(*
--报错编号0: 无报错
--报错编号1: openend Error
--报错编号2: closeract Error
*)
FUNCTION_BLOCK MFCModule
VAR_IN_OUT
	WarmHMI					:WARMStruct;
	operatorLog				:printLogModule_EX;
END_VAR
VAR_INPUT
	MFCType						:MFCType:=MFCType_Default;// 设置MFC的类型
	MFCHMItif					:MFCStruct;
	set							:BOOL:=FALSE;// 设置触发信号
	setCondition				:BOOL:=TRUE;// 设置触发条件
	clear						:BOOL:=FALSE;// 清零触发信号
	clearCondition				:BOOL:=TRUE;// 清零条件
	reset						:BOOL:=FALSE;// 复位信号
	stop						:BOOL:=FALSE;// 停止信号
	power						:BOOL:=TRUE;// TRUE--保持得电,FALSE--断开得电
	enable						:BOOL:=TRUE;// MFC禁用条件
	//ctrlMode					:ControlMode:=ControlMode.eManualCtrMode;//eManualCtrMode or eAutoCtrMode
	hmiEN						:BOOL:=TRUE;//HMI 启用条件
	
	errorDelayTime				:TIME:=T#2S;// MFC设置参数超时
	
	ACCMaxtime					:TIME:=T#2S;// MFC加速最大时间
	DCCMaxtime					:TIME:=T#2S;// MFC减速最大时间
	
	doneDelayTimeShortset		:TIME:=T#10MS;// MFC设置值到达延时_设置
	doneDelayTimeShortclear		:TIME:=T#10MS;// MFC设置值到达延时_清零
	errorID						:UDINT:=0;// MFC错误报警分配的起始ID
	nameTXT						:STRING(255):='';// MFC名字
	
	AlmAprSw					:BOOL:=FALSE;// 分子泵报警感应器信号,需要链接到实际的IO点
	
	temperatureMax				:REAL;// MFC温度报警设置值
	setFlow						:UDINT;// MFC流量设定
	maxSetValue					:REAL;// MFC流量设定上限
	minSetValue					:REAL;// MFC流量设定下限
	serialSlaveID				:UINT;// MFC ID
	serialError					:BOOL;// MFC通讯错误
	noteWTXT_set				:WSTRING(255):="";// MFC设置动作NoteTXT 中文
	noteWTXT_clear				:WSTRING(255):="";// MFC清零动作NoteTXT 中文
	
	serialExcute				:BOOL;// 通讯数据发送
	connected					:BOOL;
	connectedCount				:UDINT;
	flow					:UDINT;// 设定反馈流量值
	
	actflow					:UDINT;// 实际反馈流量值
	actflowFloat			:REAL;// 实际反馈流量值
END_VAR
VAR_OUTPUT
	note_set				:BOOL;// 设置条件不满足提示
	note_clear				:BOOL;// 清零条件不满足提示
	
	sendBusy				:BOOL;// 串口发送数据繁忙
	
	busy					:BOOL;// MFC动作Busy状态
	setbusy					:BOOL;// MFC设置动作Busy状态
	clearbusy				:BOOL;// MFC清零动作Busy状态
	done					:BOOL;// MFCdone状态
	setdone					:BOOL;// MFC设置完成
	cleardone				:BOOL;// MFC清零完成
	error					:BOOL;//  MFC error状态
	errID					:UDINT;// MFC errID
	errTXT					:STRING(255):='';//  MFC errTXT
	errWTXT					:WSTRING(255):="";//  MFC errTXT 中文
END_VAR
	
VAR	
	setErrorDelayTon		:Ton;
	setDoneDelayTon			:Ton;
	clearErrorDelayTon		:Ton;
	clearDoneDelayTon		:Ton;
	
	setTrigRAlc			    :R_Trig;//上升沿触发
	
	clearTrigRAlc			:R_Trig;//上升沿触发
	
	setTrigR1			:R_Trig;//上升沿触发
	setTrigR1_Aiko		:R_Trig;//上升沿触发
	clearRactTrigR1			:R_Trig;//上升沿触发
	resetTrigR1				:R_Trig;//上升沿触发
	stopTrigR1				:R_Trig;//上升沿触发
	powerTrigR1				:R_Trig;//上升沿触发
	
	setStep					:UINT:=0;
	clearStep				:UINT:=0;
	errorStep				:UINT:=0;
	
	resetRelayTON			:TON;
	resetRelayTONTime		:TIME:=T#2S;
	
	AccFTrig:F_TRIG;//检测加速信号下降延
	DccFTrig:F_TRIG;// 检测减速信号下降延
	noteTON_P:tON;            // 操作提示标志位延时继电器
	noteTON_N:tON;            // 操作提示标志位延时继电器
	noteRTrig_P:R_TRIG;          // 操作提示
	noteRTrig_N:R_TRIG;          // 操作提示
END_VAR

Init_ACT();
Error_ACT();
Set_ACT();
Clear_ACT();
Reset_ACT();
Error_ACT();

(*
触发缩回动作，成功触发返回TRUE，触发失败返回FALSE
*)
METHOD Act_Clear : BOOL
VAR_INPUT
END_VAR
IF enable AND clearCondition THEN// AND NOT busy
	Act_Clear:=clear:=TRUE;
ELSE
	Act_Clear:=FALSE;
END_IF
END_METHOD

(*
触发复位报警动作，成功触发返回TRUE，触发失败返回FALSE
*)
METHOD Act_Reset : BOOL
VAR_INPUT
END_VAR
Act_Reset:=reset:=TRUE;
END_METHOD

(*
触发发送动作，成功触发返回TRUE，触发失败返回FALSE
*)
METHOD Act_SerialSend : BOOL
VAR_INPUT
END_VAR
IF TRUE THEN
	Act_SerialSend:=serialExcute:=TRUE;
ELSE
	Act_SerialSend:=FALSE;
END_IF
END_METHOD

(*
触发伸出动作，成功触发返回TRUE，触发失败返回FALSE
*)
METHOD Act_Set : BOOL
VAR_INPUT
	_setpoint:UDINT;
END_VAR
IF enable AND setCondition THEN// AND NOT busy
	setFlow:=_setpoint;
	Act_Set:=set:=TRUE;
ELSE
	Act_Set:=FALSE;
END_IF
END_METHOD

(*
触发停止输出动作，成功触发返回TRUE，触发失败返回FALSE
*)
METHOD Act_Stop : BOOL
VAR_INPUT
END_VAR
Act_Stop:=stop:=TRUE;
END_METHOD

ACTION Clear_ACT:
//MFC--clear 触发
IF clear AND NOT clearCondition THEN
	note_set:=FALSE;
	note_clear:=TRUE;
END_IF
IF clear AND enable AND NOT error AND clearCondition AND NOT clearbusy AND NOT gMFCStopLoopRead THEN// AND NOT busy
	note_set:=FALSE;
	note_clear:=FALSE;
	busy:=TRUE;
	clearbusy:=TRUE;
	setbusy:=FALSE;
	set:=FALSE;
	setdone:=FALSE;
	cleardone:=FALSE;
	setStep:=0;
	clearStep:=10;
	gMFCStopLoopRead:=TRUE;
	operatorLog.append(CONCAT(nameTXT,' Clear'));
	//errorStep:=0;
END_IF
clear:=FALSE;

CASE clearStep OF
0:
	//ready
	
10:
	IF FuncModule_RS485_MFC.loopReadStep<10 OR FuncModule_RS485_MFC.loopReadStep>270 THEN
		clearErrorDelayTon(IN:=FALSE);
		clearDoneDelayTon(IN:=FALSE);
		clearStep:=20;
		setFlow:=0;
		FuncModule_RS485_MFC.Interface_Set(serialSlaveID,setFlow);
	END_IF
	
20:
	clearErrorDelayTon(IN:=(NOT FuncModule_RS485_MFC.setDone ),PT:=errorDelayTime);
	IF clearErrorDelayTon.Q THEN
		//done:=FALSE;
		setdone:=FALSE;
		cleardone:=FALSE;
		errorStep:=2;
		clearStep:=60;
		clearbusy:=FALSE;
		setbusy:=FALSE;
		RETURN;
	END_IF
	clearDoneDelayTon(IN:=FuncModule_RS485_MFC.setDone,PT:=doneDelayTimeShortclear);
	IF clearDoneDelayTon.Q THEN
		clearErrorDelayTon(IN:=FALSE);
		clearDoneDelayTon(IN:=FALSE);
		setFlow:=0;
		// send Set point
		clearStep:=30;
	END_IF
30:
	IF NOT error THEN
		busy:=FALSE;
		clearbusy:=FALSE;
		setbusy:=FALSE;
		//done:=TRUE;
		setdone:=FALSE;
		cleardone:=TRUE;
		errorStep:=0;
		clearStep:=50;
		gMFCStopLoopRead:=FALSE;
	ELSE
		busy:=FALSE;
		clearbusy:=FALSE;
		setbusy:=FALSE;
		//done:=TRUE;
		setdone:=FALSE;
		cleardone:=FALSE;
		errorStep:=3;
		clearStep:=60;
		gMFCStopLoopRead:=FALSE;
	END_IF
END_CASE
END_ACTION

ACTION Error_ACT:
CASE errorStep OF
	0:
		error:=FALSE;
		errID:=0;
		errTXT:='';
 (*
	1:
		error:=TRUE;
		errID:=errorID+errorStep;
		errTXT:=CONCAT(STR1:=nameTXT,STR2:=' Extend Error!');
		errWTXT:=WCONCAT(STR1:=TO_WSTRING(nameTXT),STR2:=" 伸出(打开)错误");
	2:
		error:=TRUE;
		errID:=errorID+errorStep;
		errTXT:=CONCAT(STR1:=nameTXT,STR2:=' Retract Error!');
		errWTXT:=WCONCAT(STR1:=TO_WSTRING(nameTXT),STR2:=" 缩回(关闭)错误");
		*)
	1..5:
		error:=TRUE;
		errID:=getErrID(errorStep);
		errTXT:=getErrTXT(errorStep);
		errWTXT:=getErrWTXT(errorStep);
END_CASE
END_ACTION

METHOD Get_Done_Clear : BOOL
VAR_INPUT
END_VAR
Get_Done_Clear:=cleardone;
END_METHOD

METHOD Get_Done_Set : BOOL
VAR_INPUT
END_VAR
Get_Done_Set:=setdone;
END_METHOD

METHOD getErrID : UDINT
VAR_INPUT
	errID					:UDINT;//取值范围1~2
END_VAR
VAR
	nErrID					:UDINT;
END_VAR
nErrID:=errorID+errID;

getErrID:=nErrID;
END_METHOD

METHOD getErrTXT : STRING(255)
VAR_INPUT
	errID					:UDINT;//取值范围1~2
END_VAR
VAR
	sErrTXT					:STRING(255);
END_VAR

CASE errID OF
	1:
		sErrTXT:=CONCAT(STR1:=nameTXT,STR2:=' Set Error!');
	2:
		sErrTXT:=CONCAT(STR1:=nameTXT,STR2:=' Clear Error!');
	3:
		sErrTXT:=CONCAT(STR1:=nameTXT,STR2:=' NormalRun Error!');
	4:
		sErrTXT:=CONCAT(STR1:=nameTXT,STR2:=' SetValue Error!');
	5:
		sErrTXT:=CONCAT(STR1:=nameTXT,STR2:=' IO Fault!');
ELSE
	sErrTXT:=CONCAT(STR1:=nameTXT,STR2:='');
END_CASE
getErrTXT:=sErrTXT;
END_METHOD

METHOD getErrWTXT : WSTRING(255)
VAR_INPUT
	errID					:UDINT;//取值范围1~16
END_VAR
VAR
	sErrTXT					:WSTRING(255);
END_VAR

CASE errID OF
	1:
		sErrTXT:=WCONCAT(STR1:=TO_WSTRING(nameTXT),STR2:="  设置 错误");
	2:
		sErrTXT:=WCONCAT(STR1:=TO_WSTRING(nameTXT),STR2:="  清零 错误");
	3:
		sErrTXT:=WCONCAT(STR1:=TO_WSTRING(nameTXT),STR2:="  正常运行出现异常情况");
	4:
		sErrTXT:=WCONCAT(STR1:=TO_WSTRING(nameTXT),STR2:="  参数设置出错");
	5:
		sErrTXT:=WCONCAT(STR1:=TO_WSTRING(nameTXT),STR2:="  IO报错");
ELSE
	sErrTXT:=WCONCAT(STR1:=TO_WSTRING(nameTXT),STR2:="");
END_CASE
getErrWTXT:=sErrTXT;
END_METHOD

ACTION Init_ACT:
done:=(cleardone OR setdone);
IF AlmAprSw THEN
	errorStep:=5;
END_IF
error:=error OR serialError OR AlmAprSw;
manualCtrl_ACT();
IF (error OR AlmAprSw OR serialError) AND flow>0.1 THEN
	stop:=TRUE;
	busy:=FALSE;
END_IF

noteTON_P(IN:=note_set,PT:=T#0.1S);
noteRTrig_P(CLK:=noteTON_P.Q);
IF noteRTrig_P.Q THEN
	//gLog_Note.append_EX(noteWTXT_Open);
	;
END_IF
noteTON_N(IN:=note_clear,PT:=T#0.1S);
noteRTrig_N(CLK:=noteTON_N.Q);
IF noteRTrig_N.Q THEN
	//gLog_Note.append_EX(noteWTXT_close);
	;
END_IF
END_ACTION

ACTION ManualCtrl_ACT:
////HMI手动控制
////IF ctrlMode=eManualCtrMode THEN
IF hmiEN THEN
	setTrigR1(CLK:=MFCHMItif.set);
	IF setTrigR1.Q THEN
		MFCHMItif.set:=FALSE;
		WarmHMI.showText:='';
		WarmHMI.showFlag:=TRUE;
		WarmHMI.showText:=CONCAT(WarmHMI.showText,'Are you sure you want ');
		WarmHMI.showText:=CONCAT(WarmHMI.showText,nameTXT);
		WarmHMI.showText:=CONCAT(WarmHMI.showText,' to Set it?');
	END_IF
	IF WarmHMI.bOK AND NOT WarmHMI.showFlag AND FIND(WarmHMI.showText,nameTXT)>0 AND FIND(WarmHMI.showText,'Set')>0 THEN
		set:=TRUE;
		WarmHMI.bOK:=FALSE;
		WarmHMI.showText:='';
	END_IF
	IF WarmHMI.bNO AND NOT WarmHMI.showFlag AND FIND(WarmHMI.showText,nameTXT)>0 AND FIND(WarmHMI.showText,'Set')>0 THEN
		WarmHMI.bNO:=FALSE;
		MFCHMItif.set:=FALSE;
		WarmHMI.showText:='';
	END_IF
	clearTrigRAlc(CLK:=MFCHMItif.clear);
	IF clearTrigRAlc.Q THEN
		MFCHMItif.clear:=FALSE;
		WarmHMI.showText:='';
		WarmHMI.showFlag:=TRUE;
		WarmHMI.showText:=CONCAT(WarmHMI.showText,'Are you sure you want to Clear the ');
		WarmHMI.showText:=CONCAT(WarmHMI.showText,nameTXT);
		WarmHMI.showText:=CONCAT(WarmHMI.showText,' `Par?');
	END_IF
	IF WarmHMI.bOK AND NOT WarmHMI.showFlag AND FIND(WarmHMI.showText,nameTXT)>0 AND FIND(WarmHMI.showText,'Clear')>0 THEN
		clear:=TRUE;
		WarmHMI.bOK:=FALSE;
		WarmHMI.showText:='';
	END_IF
	IF WarmHMI.bNO AND NOT WarmHMI.showFlag AND FIND(WarmHMI.showText,nameTXT)>0 AND FIND(WarmHMI.showText,'Clear')>0 THEN
		WarmHMI.bNO:=FALSE;
		MFCHMItif.clear:=FALSE;
		WarmHMI.showText:='';
	END_IF
END_IF
END_ACTION

ACTION Reset_ACT:
IF reset THEN
	note_set:=FALSE;
	note_clear:=FALSE;
	setStep:=0;
	clearStep:=0;
	errorStep:=0;
	reset:=FALSE;
END_IF
//resetRelayTON(IN:=resetRelay , PT:=resetRelayTONTime);
//IF resetRelayTON.Q THEN
//	openStep:=0;
//	closeStep:=0;
//	errorStep:=0;
//	busy:=FALSE;
//	resetRelay:=FALSE;
//END_IF

//IF stop THEN
//	note_open:=FALSE;
//	note_close:=FALSE;
//	stop:=FALSE;
//	openRelay:=FALSE;
//	closeRelay:=FALSE;
//	//无自锁检测说法，直接停
//	openStep:=0;
//	closeStep:=0;
//END_IF
END_ACTION

ACTION Serial_Act:
//(*
// *功能块的作用，把 TxBuffer 缓存区的数据经过 Process Data 的 ComOut 发送出去，
// *而把 ComIn 中的数据接收到 RxBuffer。引用这个功能块的程序执行周期越短，
// *数据交换的效率就越高，所以这段程序应该放在快速任务中作为 Backgroud 代码无条件执行。
//*)
//COMportControl(
//	Mode:= SERIALLINEMODE_KL6_22B_STANDARD, 
//	pComIn:= ADR(COMin), 
//	pComOut:= ADR(COMout), 
//	SizeComIn:= SIZEOF(COMin), 
//	Error=> , 
//	ErrorID=> , 
//	TxBuffer:= TxBuffer_TMP, 
//	RxBuffer:= RxBuffer_TMP );
//IF receive1.Error <> COMERROR_NOERROR THEN
//	serialRecError:=TRUE;
//END_IF
//receive1(
//	pPrefix:= , 
//	LenPrefix:= , 
//	pSuffix:= , 
//	LenSuffix:= , 
//	pReceiveData:= ADR(arr_RcvData), 
//	SizeReceiveData:= 100, 
//	Timeout:= T#100MS, //临时设置成10S调试用
//	Reset:= , 
//	DataReceived=> , 
//	busy=> , 
//	Error=> , 
//	RxTimeout=> , 
//	LenReceiveData=> , 
//	RXbuffer:= RxBuffer_TMP);
////testReal:=BYTE_TO_REAL(arr_RcvData_Temp);
//CASE serialStep OF
//	0:
//	IF enableSerial AND serialExcute THEN
//		serialExcute:=FALSE;
//		IF NOT serialBusy THEN
//			serialStep:=10;
//			serialBusy:=TRUE;
//			serialDone:=FALSE;
//			serialError:=FALSE;
//			serialTimeOut:=FALSE;
//			serialRecError:=FALSE;
//			receive1(//复位
//				pPrefix:= , 
//				LenPrefix:= , 
//				pSuffix:= , 
//				LenSuffix:= , 
//				pReceiveData:= , 
//				SizeReceiveData:=, 
//				Timeout:= T#300MS, 
//				Reset:= , 
//				DataReceived=> , 
//				busy=> , 
//				Error=> , 
//				RxTimeout=> , 
//				LenReceiveData=> , 
//				RXbuffer:= RxBuffer_TMP);
//		END_IF
//	END_IF
//	Timer1(IN:= FALSE);
//	;
//	10:
//		//第二和第三位代表ID号
//		arr_SendData[1]	:=16#40;
//		IF serialSlaveID>9 THEN
//			arr_SendData[2]	:=F_ToASC(str:='0');
//			arr_SendData[3]	:=F_ToASC(str:=(UINT_TO_STRING(serialSlaveID)));
//		ELSE
//			arr_SendData[2]	:=F_ToASC(str:=(UINT_TO_STRING(serialSlaveID/10)));
//			arr_SendData[3]	:=F_ToASC(str:=(UINT_TO_STRING(serialSlaveID MOD 10)));
//		END_IF
//		arr_SendData[4]:=16#02;
//		arr_SendData[5]:=16#30;
//		arr_SendData[6]:=16#30;
//		arr_SendData[7]:=16#31;
//		arr_SendData[8]:=16#3F;
//		arr_SendData[9]:=16#5B;
//		arr_SendData[10]:=16#03;
//		arr_SendData[11]:=16#AB;
//		serialStep:=100;
//	100:
//		send1(
//			pSendData:= ADR(arr_SendData), 
//			Length:= nSendByteLength, 
//			Busy=> , 
//			Error=> , 
//			TXbuffer:= TxBuffer_TMP);
//		serialStep:=serialStep+20;
//	110:
//		Timer1(IN:= NOT timer1.q, PT:=T#00MS);
//		IF Timer1.Q THEN
//			serialStep:=serialStep+10;
//			Timer1(IN:= FALSE);
//		END_IF
//	120:
//		Timer1(IN:= NOT timer1.q, PT:=T#3000MS);
//		IF Timer1.Q THEN
//			serialStep:=6000;
//			Timer1(IN:= FALSE);
//			serialTimeOut:=TRUE;
//			RETURN;
//		END_IF
//		IF receive1.DataReceived THEN
//			Timer1(IN:= FALSE);
//			serialTimeOut:=FALSE;
//			serialStep:=200;
//		END_IF
//		IF receive1.Error <> COMERROR_NOERROR THEN
//			serialRecError:=TRUE;
//		END_IF
//	200://数据处理
//		arr_RcvData_Temp:=arr_RcvData;
//		arr_RcvData:=arr_RcvData_Clear;
//		serialStep:=serialStep+10;
//	210:
//		//第二和第三位代表ID号;看情况决定是否需要判断节点反馈的节点号
//		IF arr_RcvData_Temp[12]=arr_SendData[9] AND arr_RcvData_Temp[2]=arr_SendData[2] AND arr_RcvData_Temp[3]=arr_SendData[3] THEN
//			serialStep:=serialStep+10;
//			serialRecError:=FALSE;
//		ELSE//数据接线错误
//			serialStep:=6000;
//			serialRecError:=TRUE;
//		END_IF
//	220:
//		//数据转换
//		serialStep:=300;
//	;
//	300:
//		strTemp:='';
//		strTemp:=CONCAT(strTemp,F_TOCHR(arr_RcvData_Temp[47]));
//		strTemp:=CONCAT(strTemp,F_TOCHR(arr_RcvData_Temp[48]));
//		strTemp:=CONCAT(strTemp,F_TOCHR(arr_RcvData_Temp[49]));
//		strTemp:=CONCAT(strTemp,F_TOCHR(arr_RcvData_Temp[50]));
//		temperature:=STRING_TO_UINT(strTemp)*1.0;
//		strTemp:='';
//		strTemp:=CONCAT(strTemp,F_TOCHR(arr_RcvData_Temp[53]));
//		strTemp:=CONCAT(strTemp,F_TOCHR(arr_RcvData_Temp[54]));
//		currentTemp:=STRING_TO_INT(strTemp);
//		current:=INT_TO_REAL(currentTemp)/10.0;// 1位小数
//		strTemp:='';
//		strTemp:=CONCAT(strTemp,F_TOCHR(arr_RcvData_Temp[61]));
//		strTemp:=CONCAT(strTemp,F_TOCHR(arr_RcvData_Temp[62]));
//		strTemp:=CONCAT(strTemp,F_TOCHR(arr_RcvData_Temp[63]));
//		strTemp:=CONCAT(strTemp,F_TOCHR(arr_RcvData_Temp[64]));
//		speed:=STRING_TO_UINT(strTemp)*1.0;
//		serialStep:=5000;
//	;
//	5000://done
//		serialBusy:=FALSE;
//		serialDone:=TRUE;
//		serialError:=FALSE;
//		serialStep:=0;
//	;
//	6000://error
//		serialBusy:=FALSE;
//		serialDone:=FALSE;
//		serialError:=TRUE;
//		serialStep:=0;
//	;
	
//END_CASE
////arr_Temp[1]:=arr_RcvData_Temp[48];
////arr_Temp[2]:=arr_RcvData_Temp[47];
////MEMMOVE(ADR(temperatureTemp),ADR(arr_Temp[1]),2);// 2个字节
////temperature:=DINT_TO_REAL(temperatureTemp);
////MEMMOVE(ADR(currentTemp),ADR(arr_RcvData_Temp[53]),1);// 1个字节
////current:=INT_TO_REAL(currentTemp)/1.0;// 1位小数
////arr_Temp1[1]:=arr_RcvData_Temp[62];
////arr_Temp1[2]:=arr_RcvData_Temp[61];
////MEMMOVE(ADR(speedTemp),ADR(arr_Temp1[1]),2);// 2个字节
////speed:=DINT_TO_REAL(speedTemp);
////speed:=speed*60.0;
////IF enableSerial THEN//启用
////	;
////	 //字符串方式
////	 (*//3000ms发送一次
////	Timer1(IN:= NOT timer1.q, PT:=T#3000MS , Q=> , ET=> );
////	IF timer1.Q THEN
////		SEND1(
////			SendString:=_sendString ,
////			TXbuffer:=TxBuffer_TMP ,
////			Busy=> ,
////			Error=> );
////	END_IF
	 
////	//接收
////	Receive1(
////		Timeout:= t#100ms,
////		ReceivedString:=_receive1string ,
////		RXbuffer:=RxBuffer_TMP , );
	 
////	//保存上一个周期接收的字符
////	IF Receive1.Busy THEN
////		_recvLast:=_receive1string;
////	END_IF*)
////END_IF
END_ACTION

ACTION Set_ACT:
//MFC--set 触发
IF set AND NOT setCondition THEN
	note_clear:=FALSE;
	note_set:=TRUE;
END_IF
IF set AND enable AND NOT error AND setCondition AND NOT setbusy AND NOT gMFCStopLoopRead THEN// AND NOT busy
	note_set:=FALSE;
	note_clear:=FALSE;
	busy:=TRUE;
	setbusy:=TRUE;
	clearbusy:=FALSE;
	set:=FALSE;
	setdone:=FALSE;
	cleardone:=FALSE;
	setStep:=10;
	clearStep:=0;
	gMFCStopLoopRead:=TRUE;
	operatorLog.append(CONCAT(CONCAT(nameTXT,' Set '),UDINT_TO_STRING(setFlow)));
	//errorStep:=0;
END_IF
set:=FALSE;

CASE setStep OF
0:
	//ready

10:
 	IF FuncModule_RS485_MFC.loopReadStep<10 OR FuncModule_RS485_MFC.loopReadStep>270 THEN
		setErrorDelayTon(IN:=FALSE);
		setDoneDelayTon(IN:=FALSE);
		IF (UDINT_TO_REAL(setFlow)<=maxSetValue AND UDINT_TO_REAL(setFlow)>=minSetValue) THEN
			setStep:=20;
			FuncModule_RS485_MFC.Interface_Set(serialSlaveID,setFlow);
		ELSE
			setdone:=FALSE;
			cleardone:=FALSE;
			setStep:=60;
			gMFCStopLoopRead:=FALSE;
			errorStep:=4;
			setFlow:=flow;
			clearbusy:=FALSE;
			setbusy:=FALSE;
			setDoneDelayTon(IN:=FALSE);
			setErrorDelayTon(IN:=FALSE);
		END_IF
	END_IF
20:
	setErrorDelayTon(IN:=(NOT FuncModule_RS485_MFC.setDone ),PT:=errorDelayTime);
	IF setErrorDelayTon.Q THEN
		//done:=FALSE;
		setdone:=FALSE;
		cleardone:=FALSE;
		errorStep:=1;
		setStep:=60;
		gMFCStopLoopRead:=FALSE;
		clearbusy:=FALSE;
		setbusy:=FALSE;
		RETURN;
	END_IF
	setDoneDelayTon(IN:=FuncModule_RS485_MFC.setDone,PT:=doneDelayTimeShortset);
	IF setDoneDelayTon.Q THEN
		setErrorDelayTon(IN:=FALSE);
		setDoneDelayTon(IN:=FALSE);
		setStep:=30;
	END_IF
30:
	IF NOT error THEN
		busy:=FALSE;
		clearbusy:=FALSE;
		setbusy:=FALSE;
		//done:=TRUE;
		cleardone:=FALSE;
		setdone:=TRUE;
		errorStep:=0;
		setStep:=50;
		gMFCStopLoopRead:=FALSE;
	ELSE
		busy:=FALSE;
		clearbusy:=FALSE;
		setbusy:=FALSE;
		//done:=TRUE;
		setdone:=FALSE;
		cleardone:=FALSE;
		errorStep:=3;
		setFlow:=flow;
		setStep:=60;
		gMFCStopLoopRead:=FALSE;
	END_IF

END_CASE
END_ACTION

ACTION VersionLog:
(*
版本: V1.0.0.0
说明:
	1. 首个版本
	2. 含普通分子泵\泵组类型的控制
	3. 可配置是否有到位信号, 以及到位稳定时间
*)
END_ACTION

END_FUNCTION_BLOCK

(* stored: Version 1.1.0.1, ProductVersion 3.1.4024.4
   POU MFCModule: Id {b84dba2e-dfd5-42c5-b4c6-6aae2a5c9dcd}, SpecialFunc None
   Folder Error: Id {5da1e154-2126-43da-ada3-209eff6eaa3a}
   Folder Private: Id {588d8152-aeea-4a3f-8869-c07f16492789}
   Method Act_Clear: Id {882ba459-a59a-408c-a2e4-3ee5cf6e3fbf}
   Method Act_Reset: Id {67b5c228-3b68-46ef-b237-8797f45b6eaa}
   Method Act_SerialSend: Id {b079b726-39dd-4cf1-9715-b8f31e870381}
   Method Act_Set: Id {7c7db399-199e-4bc6-8ece-2d6de3b0052d}
   Method Act_Stop: Id {b2707cc9-33d5-452e-a6f9-dfe1213df716}
   Action Clear_ACT: Id {4bb9c453-968b-43a6-8252-1dc5b468227f}
   Action Error_ACT: Id {f216cb17-e9f0-419d-b79f-fec08e94dfb5}
   Method Get_Done_Clear: Id {d42b1037-74c1-4e3f-8a37-ec2aeae19903}
   Method Get_Done_Set: Id {6ea7b300-5a25-48cc-9c22-bffea72edd85}
   Method getErrID: Id {15d57b93-4f8f-4fe1-a21c-660da2d7b58a}
   Method getErrTXT: Id {f92480f2-2850-4975-9926-d01361c9c81e}
   Method getErrWTXT: Id {5cd5dc0c-66dc-4067-b622-779890a52302}
   Action Init_ACT: Id {79d7cdf0-39b5-4224-b662-16ad89b57235}
   Action ManualCtrl_ACT: Id {d64d2857-6c72-4464-b7b6-764c2d372a14}
   Action Reset_ACT: Id {acc7fd02-8282-4600-96b6-508b97e8ea14}
   Action Serial_Act: Id {910a0794-ece2-4050-84b7-e0f45f138426}
   Action Set_ACT: Id {c6df1d36-5b0d-4093-ac0a-181f047cc7c7}
   Action VersionLog: Id {21b67494-c9b5-4739-bd31-a7ffe7222174} *)
